# B&R Automation Studio project ProcessPointsTest
Automation Studio 4.11.6.26 SP; technology packages: mappMotion 5.23.1

## Configuration Config1

CPU PC_any, AutomationRuntime D4.92, Build 4.1.2, Safety 0.0, Vc V4.72.5

### Task classes (Cpu.sw)
```
Cyclic#1 (cycle 1600 us, tolerance 0 us):
  Program <- Program.prg
DataObjects: McAcpSys
NcDataObjects: McDriveLog
Binaries: arsvcreg, udbdef, McAcpDrv, arflatprv, arcoal, FWRules, TCData, McAcpSim, ashwd, ashwac, Points, User, Machine, sysconf, ShuttleCon, asfw, arconfig, ShuttleSim, iomap, Sectors, Role
Libraries: McBase, McAxis, McAcpTrak, MpBase, MpAxis, McAcpAx, standard, AsBrStr, runtime, asieccon, powerlnk, astime, fileio, sys_lib, asepl
```

### Hardware
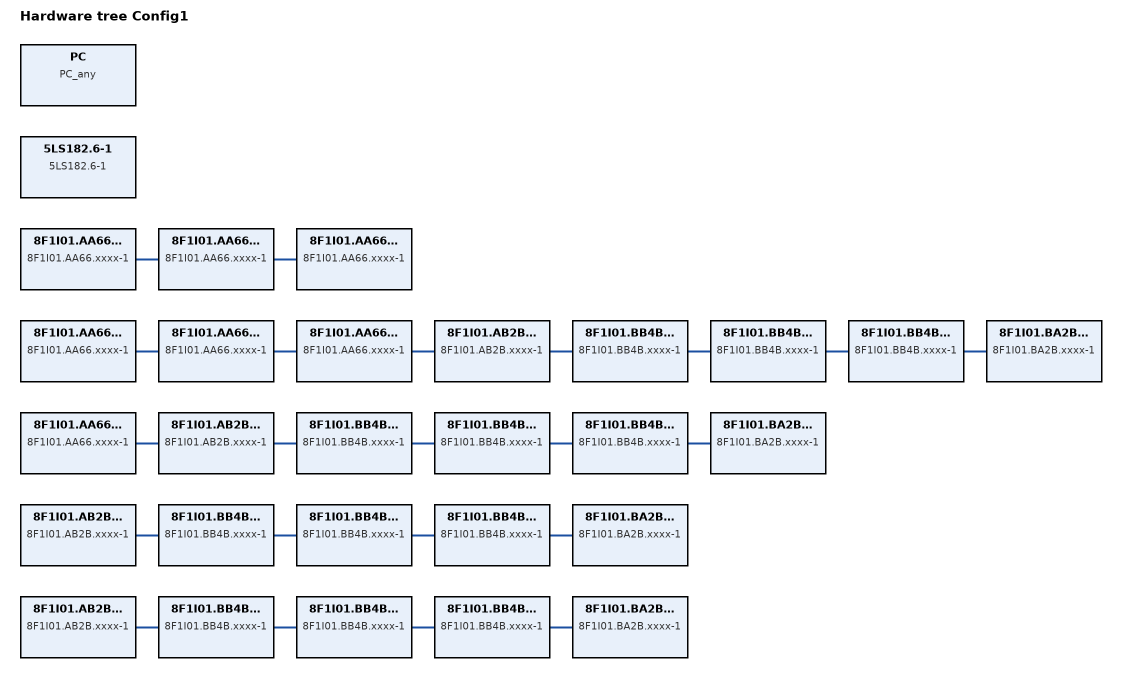
```
5LS182.6-1 : 5LS182.6-1 v1.3.1.0  [PLK2 -> 8F1I01.AA66.xxxx-1f.PLK3 [Cable Type=PowerlinkCable, Length=10, Version=1.0.0.3]; SL -> PC.SL1]
  Connector IF1:
    CycleTime = 800
  Supervision = off
8F1I01.AA66.xxxx-1 : 8F1I01.AA66.xxxx-1 v1.0.0.2  [PLK1 -> 8F1I01.BA2B.xxxx-1.PLK2 (NodeNumber=6) [Cable Type=PowerlinkCable, Length=10, Version=1.0.0.3]; PLK2 -> 8F1I01.AA66.xxxx-1a.PLK1 (NodeNumber=6) [Cable Type=PowerlinkCable, Length=10, Version=1.0.0.3]]
  DriveConfiguration:
    McTypeID = LLMConfig
  DriveConfiguration/Segment:
    Shape = STRAIGHT660
    SegmentReference = A06
    SegmentSectorDirection = Positive
    ElongationCompensation = UseAssemblySetting
    StopReaction = UseAssemblySetting
    SpeedFilter = UseAssemblySetting
    PositionControllerLagMonitor = UseAssemblySetting
8F1I01.AA66.xxxx-1a : 8F1I01.AA66.xxxx-1 v1.0.0.2  [PLK1 -> 8F1I01.AA66.xxxx-1.PLK2 (NodeNumber=7) [Cable Type=PowerlinkCable, Length=10, Version=1.0.0.3]; PLK2 -> 8F1I01.AA66.xxxx-1b.PLK1 (NodeNumber=7) [Cable Type=PowerlinkCable, Length=10, Version=1.0.0.3]]
  DriveConfiguration:
    McTypeID = LLMConfig
  DriveConfiguration/Segment:
    Shape = STRAIGHT660
    SegmentReference = A07
    SegmentSectorDirection = Positive
    ElongationCompensation = UseAssemblySetting
    StopReaction = UseAssemblySetting
    SpeedFilter = UseAssemblySetting
    PositionControllerLagMonitor = UseAssemblySetting
8F1I01.AA66.xxxx-1b : 8F1I01.AA66.xxxx-1 v1.0.0.2  [PLK1 -> 8F1I01.AA66.xxxx-1a.PLK2 (NodeNumber=8) [Cable Type=PowerlinkCable, Length=10, Version=1.0.0.3]]
  DriveConfiguration:
    McTypeID = LLMConfig
  DriveConfiguration/Segment:
    Shape = STRAIGHT660
    SegmentReference = A08
    SegmentSectorDirection = Positive
    ElongationCompensation = UseAssemblySetting
    StopReaction = UseAssemblySetting
    SpeedFilter = UseAssemblySetting
    PositionControllerLagMonitor = UseAssemblySetting
8F1I01.AA66.xxxx-1c : 8F1I01.AA66.xxxx-1 v1.0.0.2  [PLK1 -> 8F1I01.BA2B.xxxx-1a.PLK2 (NodeNumber=14) [Cable Type=PowerlinkCable, Length=10, Version=1.0.0.3]; PLK2 -> 8F1I01.AA66.xxxx-1d.PLK1 (NodeNumber=14) [Cable Type=PowerlinkCable, Length=10, Version=1.0.0.3]]
  DriveConfiguration:
    McTypeID = LLMConfig
  DriveConfiguration/Segment:
    Shape = STRAIGHT660
    SegmentReference = A14
    SegmentSectorDirection = Positive
    ElongationCompensation = UseAssemblySetting
    StopReaction = UseAssemblySetting
    SpeedFilter = UseAssemblySetting
    PositionControllerLagMonitor = UseAssemblySetting
8F1I01.AA66.xxxx-1d : 8F1I01.AA66.xxxx-1 v1.0.0.2  [PLK1 -> 8F1I01.AA66.xxxx-1c.PLK2 (NodeNumber=15) [Cable Type=PowerlinkCable, Length=10, Version=1.0.0.3]; PLK2 -> 8F1I01.AA66.xxxx-1e.PLK1 (NodeNumber=15) [Cable Type=PowerlinkCable, Length=10, Version=1.0.0.3]]
  DriveConfiguration:
    McTypeID = LLMConfig
  DriveConfiguration/Segment:
    Shape = STRAIGHT660
    SegmentReference = A15
    SegmentSectorDirection = Positive
    ElongationCompensation = UseAssemblySetting
    StopReaction = UseAssemblySetting
    SpeedFilter = UseAssemblySetting
    PositionControllerLagMonitor = UseAssemblySetting
8F1I01.AA66.xxxx-1e : 8F1I01.AA66.xxxx-1 v1.0.0.2  [PLK1 -> 8F1I01.AA66.xxxx-1d.PLK2 (NodeNumber=16) [Cable Type=PowerlinkCable, Length=10, Version=1.0.0.3]; PLK2 -> 8F1I01.AB2B.xxxx-1.PLK1 (NodeNumber=16) [Cable Type=PowerlinkCable, Length=10, Version=1.0.0.3]]
  DriveConfiguration:
    McTypeID = LLMConfig
  DriveConfiguration/Segment:
    Shape = STRAIGHT660
    SegmentReference = A16
    SegmentSectorDirection = Positive
    ElongationCompensation = UseAssemblySetting
    StopReaction = UseAssemblySetting
    SpeedFilter = UseAssemblySetting
    PositionControllerLagMonitor = UseAssemblySetting
8F1I01.AA66.xxxx-1f : 8F1I01.AA66.xxxx-1 v1.0.0.2  [PLK1 -> 8F1I01.BA2B.xxxx-1c.PLK2 (NodeNumber=17) [Cable Type=PowerlinkCable, Length=10, Version=1.0.0.3]; PLK2 -> 8F1I01.AB2B.xxxx-1b.PLK1 (NodeNumber=17) [Cable Type=PowerlinkCable, Length=10, Version=1.0.0.3]; PLK3 -> 5LS182.6-1.PLK2 (NodeNumber=17) [Cable Type=PowerlinkCable, Length=10, Version=1.0.0.3]]
  DriveConfiguration:
    McTypeID = LLMConfig
  DriveConfiguration/Segment:
    Shape = STRAIGHT660
    SegmentReference = B06
    SegmentSectorDirection = Positive
    ElongationCompensation = UseAssemblySetting
    StopReaction = UseAssemblySetting
    SpeedFilter = UseAssemblySetting
    PositionControllerLagMonitor = UseAssemblySetting
8F1I01.AB2B.xxxx-1 : 8F1I01.AB2B.xxxx-1 v1.0.0.2  [PLK1 -> 8F1I01.AA66.xxxx-1e.PLK2 (NodeNumber=1) [Cable Type=PowerlinkCable, Length=10, Version=1.0.0.3]; PLK2 -> 8F1I01.BB4B.xxxx-1.PLK1 (NodeNumber=1) [Cable Type=PowerlinkCable, Length=10, Version=1.0.0.3]; PLK3 -> 5LS182.6-1.IF1 (NodeNumber=1) [Cable Type=PowerlinkCable, Length=10, Version=1.0.0.3]]
  DriveConfiguration:
    McTypeID = LLMConfig
  DriveConfiguration/Segment:
    Shape = STRAIGHT105_TO_CIRCULAR
    SegmentReference = A01
    SegmentSectorDirection = Positive
    ElongationCompensation = UseAssemblySetting
    StopReaction = UseAssemblySetting
    SpeedFilter = UseAssemblySetting
    PositionControllerLagMonitor = UseAssemblySetting
8F1I01.AB2B.xxxx-1a : 8F1I01.AB2B.xxxx-1 v1.0.0.2  [PLK2 -> 8F1I01.BB4B.xxxx-1c.PLK1 (NodeNumber=9) [Cable Type=PowerlinkCable, Length=10, Version=1.0.0.3]]
  DriveConfiguration:
    McTypeID = LLMConfig
  DriveConfiguration/Segment:
    Shape = STRAIGHT105_TO_CIRCULAR
    SegmentReference = A09
    SegmentSectorDirection = Positive
    ElongationCompensation = UseAssemblySetting
    StopReaction = UseAssemblySetting
    SpeedFilter = UseAssemblySetting
    PositionControllerLagMonitor = UseAssemblySetting
8F1I01.AB2B.xxxx-1b : 8F1I01.AB2B.xxxx-1 v1.0.0.2  [PLK1 -> 8F1I01.AA66.xxxx-1f.PLK2 (NodeNumber=18) [Cable Type=PowerlinkCable, Length=10, Version=1.0.0.3]; PLK2 -> 8F1I01.BB4B.xxxx-1f.PLK1 (NodeNumber=18) [Cable Type=PowerlinkCable, Length=10, Version=1.0.0.3]]
  DriveConfiguration:
    McTypeID = LLMConfig
  DriveConfiguration/Segment:
    Shape = STRAIGHT105_TO_CIRCULAR
    SegmentReference = B07
    SegmentSectorDirection = Positive
    ElongationCompensation = UseAssemblySetting
    StopReaction = UseAssemblySetting
    SpeedFilter = UseAssemblySetting
    PositionControllerLagMonitor = UseAssemblySetting
8F1I01.AB2B.xxxx-1c : 8F1I01.AB2B.xxxx-1 v1.0.0.2  [PLK2 -> 8F1I01.BB4B.xxxx-1k.PLK1 (NodeNumber=27) [Cable Type=PowerlinkCable, Length=10, Version=1.0.0.3]]
  DriveConfiguration:
    McTypeID = LLMConfig
  DriveConfiguration/Segment:
    Shape = STRAIGHT105_TO_CIRCULAR
    SegmentReference = B01
    SegmentSectorDirection = Positive
    ElongationCompensation = UseAssemblySetting
    StopReaction = UseAssemblySetting
    SpeedFilter = UseAssemblySetting
    PositionControllerLagMonitor = UseAssemblySetting
8F1I01.BA2B.xxxx-1 : 8F1I01.BA2B.xxxx-1 v1.0.0.2  [PLK1 -> 8F1I01.BB4B.xxxx-1b.PLK2 (NodeNumber=5) [Cable Type=PowerlinkCable, Length=10, Version=1.0.0.3]; PLK2 -> 8F1I01.AA66.xxxx-1.PLK1 (NodeNumber=5) [Cable Type=PowerlinkCable, Length=10, Version=1.0.0.3]]
  DriveConfiguration:
    McTypeID = LLMConfig
  DriveConfiguration/Segment:
    Shape = CIRCULAR_TO_STRAIGHT105
    SegmentReference = A05
    SegmentSectorDirection = Positive
    ElongationCompensation = UseAssemblySetting
    StopReaction = UseAssemblySetting
    SpeedFilter = UseAssemblySetting
    PositionControllerLagMonitor = UseAssemblySetting
8F1I01.BA2B.xxxx-1a : 8F1I01.BA2B.xxxx-1 v1.0.0.2  [PLK1 -> 8F1I01.BB4B.xxxx-1e.PLK2 (NodeNumber=13) [Cable Type=PowerlinkCable, Length=10, Version=1.0.0.3]; PLK2 -> 8F1I01.AA66.xxxx-1c.PLK1 (NodeNumber=13) [Cable Type=PowerlinkCable, Length=10, Version=1.0.0.3]]
  DriveConfiguration:
    McTypeID = LLMConfig
  DriveConfiguration/Segment:
    Shape = CIRCULAR_TO_STRAIGHT105
    SegmentReference = A13
    SegmentSectorDirection = Positive
    ElongationCompensation = UseAssemblySetting
    StopReaction = UseAssemblySetting
    SpeedFilter = UseAssemblySetting
    PositionControllerLagMonitor = UseAssemblySetting
8F1I01.BA2B.xxxx-1b : 8F1I01.BA2B.xxxx-1 v1.0.0.2  [PLK1 -> 8F1I01.BB4B.xxxx-1h.PLK2 (NodeNumber=22) [Cable Type=PowerlinkCable, Length=10, Version=1.0.0.3]]
  DriveConfiguration:
    McTypeID = LLMConfig
  DriveConfiguration/Segment:
    Shape = CIRCULAR_TO_STRAIGHT105
    SegmentReference = B11
    SegmentSectorDirection = Positive
    ElongationCompensation = UseAssemblySetting
    StopReaction = UseAssemblySetting
    SpeedFilter = UseAssemblySetting
    PositionControllerLagMonitor = UseAssemblySetting
8F1I01.BA2B.xxxx-1c : 8F1I01.BA2B.xxxx-1 v1.0.0.2  [PLK1 -> 8F1I01.BB4B.xxxx-1i.PLK2 (NodeNumber=23) [Cable Type=PowerlinkCable, Length=10, Version=1.0.0.3]; PLK2 -> 8F1I01.AA66.xxxx-1f.PLK1 (NodeNumber=23) [Cable Type=PowerlinkCable, Length=10, Version=1.0.0.3]]
  DriveConfiguration:
    McTypeID = LLMConfig
  DriveConfiguration/Segment:
    Shape = CIRCULAR_TO_STRAIGHT105
    SegmentReference = B05
    SegmentSectorDirection = Positive
    ElongationCompensation = UseAssemblySetting
    StopReaction = UseAssemblySetting
    SpeedFilter = UseAssemblySetting
    PositionControllerLagMonitor = UseAssemblySetting
8F1I01.BB4B.xxxx-1 : 8F1I01.BB4B.xxxx-1 v1.0.0.2  [PLK1 -> 8F1I01.AB2B.xxxx-1.PLK2 (NodeNumber=2) [Cable Type=PowerlinkCable, Length=10, Version=1.0.0.3]; PLK2 -> 8F1I01.BB4B.xxxx-1a.PLK1 (NodeNumber=2) [Cable Type=PowerlinkCable, Length=10, Version=1.0.0.3]]
  DriveConfiguration:
    McTypeID = LLMConfig
  DriveConfiguration/Segment:
    Shape = CIRCULAR
    SegmentReference = A02
    SegmentSectorDirection = Positive
    ElongationCompensation = UseAssemblySetting
    StopReaction = UseAssemblySetting
    SpeedFilter = UseAssemblySetting
    PositionControllerLagMonitor = UseAssemblySetting
8F1I01.BB4B.xxxx-1a : 8F1I01.BB4B.xxxx-1 v1.0.0.2  [PLK1 -> 8F1I01.BB4B.xxxx-1.PLK2 (NodeNumber=3) [Cable Type=PowerlinkCable, Length=10, Version=1.0.0.3]; PLK2 -> 8F1I01.BB4B.xxxx-1b.PLK1 (NodeNumber=3) [Cable Type=PowerlinkCable, Length=10, Version=1.0.0.3]]
  DriveConfiguration:
    McTypeID = LLMConfig
  DriveConfiguration/Segment:
    Shape = CIRCULAR
    SegmentReference = A03
    SegmentSectorDirection = Positive
    ElongationCompensation = UseAssemblySetting
    StopReaction = UseAssemblySetting
    SpeedFilter = UseAssemblySetting
    PositionControllerLagMonitor = UseAssemblySetting
8F1I01.BB4B.xxxx-1b : 8F1I01.BB4B.xxxx-1 v1.0.0.2  [PLK1 -> 8F1I01.BB4B.xxxx-1a.PLK2 (NodeNumber=4) [Cable Type=PowerlinkCable, Length=10, Version=1.0.0.3]; PLK2 -> 8F1I01.BA2B.xxxx-1.PLK1 (NodeNumber=4) [Cable Type=PowerlinkCable, Length=10, Version=1.0.0.3]]
  DriveConfiguration:
    McTypeID = LLMConfig
  DriveConfiguration/Segment:
    Shape = CIRCULAR
    SegmentReference = A04
    SegmentSectorDirection = Positive
    ElongationCompensation = UseAssemblySetting
    StopReaction = UseAssemblySetting
    SpeedFilter = UseAssemblySetting
    PositionControllerLagMonitor = UseAssemblySetting
8F1I01.BB4B.xxxx-1c : 8F1I01.BB4B.xxxx-1 v1.0.0.2  [PLK1 -> 8F1I01.AB2B.xxxx-1a.PLK2 (NodeNumber=10) [Cable Type=PowerlinkCable, Length=10, Version=1.0.0.3]; PLK2 -> 8F1I01.BB4B.xxxx-1d.PLK1 (NodeNumber=10) [Cable Type=PowerlinkCable, Length=10, Version=1.0.0.3]]
  DriveConfiguration:
    McTypeID = LLMConfig
  DriveConfiguration/Segment:
    Shape = CIRCULAR
    SegmentReference = A10
    SegmentSectorDirection = Positive
    ElongationCompensation = UseAssemblySetting
    StopReaction = UseAssemblySetting
    SpeedFilter = UseAssemblySetting
    PositionControllerLagMonitor = UseAssemblySetting
8F1I01.BB4B.xxxx-1d : 8F1I01.BB4B.xxxx-1 v1.0.0.2  [PLK1 -> 8F1I01.BB4B.xxxx-1c.PLK2 (NodeNumber=11) [Cable Type=PowerlinkCable, Length=10, Version=1.0.0.3]; PLK2 -> 8F1I01.BB4B.xxxx-1e.PLK1 (NodeNumber=11) [Cable Type=PowerlinkCable, Length=10, Version=1.0.0.3]]
  DriveConfiguration:
    McTypeID = LLMConfig
  DriveConfiguration/Segment:
    Shape = CIRCULAR
    SegmentReference = A11
    SegmentSectorDirection = Positive
    ElongationCompensation = UseAssemblySetting
    StopReaction = UseAssemblySetting
    SpeedFilter = UseAssemblySetting
    PositionControllerLagMonitor = UseAssemblySetting
8F1I01.BB4B.xxxx-1e : 8F1I01.BB4B.xxxx-1 v1.0.0.2  [PLK1 -> 8F1I01.BB4B.xxxx-1d.PLK2 (NodeNumber=12) [Cable Type=PowerlinkCable, Length=10, Version=1.0.0.3]; PLK2 -> 8F1I01.BA2B.xxxx-1a.PLK1 (NodeNumber=12) [Cable Type=PowerlinkCable, Length=10, Version=1.0.0.3]]
  DriveConfiguration:
    McTypeID = LLMConfig
  DriveConfiguration/Segment:
    Shape = CIRCULAR
    SegmentReference = A12
    SegmentSectorDirection = Positive
    ElongationCompensation = UseAssemblySetting
    StopReaction = UseAssemblySetting
    SpeedFilter = UseAssemblySetting
    PositionControllerLagMonitor = UseAssemblySetting
8F1I01.BB4B.xxxx-1f : 8F1I01.BB4B.xxxx-1 v1.0.0.2  [PLK1 -> 8F1I01.AB2B.xxxx-1b.PLK2 (NodeNumber=19) [Cable Type=PowerlinkCable, Length=10, Version=1.0.0.3]; PLK2 -> 8F1I01.BB4B.xxxx-1g.PLK1 (NodeNumber=19) [Cable Type=PowerlinkCable, Length=10, Version=1.0.0.3]]
  DriveConfiguration:
    McTypeID = LLMConfig
  DriveConfiguration/Segment:
    Shape = CIRCULAR
    SegmentReference = B08
    SegmentSectorDirection = Positive
    ElongationCompensation = UseAssemblySetting
    StopReaction = UseAssemblySetting
    SpeedFilter = UseAssemblySetting
    PositionControllerLagMonitor = UseAssemblySetting
8F1I01.BB4B.xxxx-1g : 8F1I01.BB4B.xxxx-1 v1.0.0.2  [PLK1 -> 8F1I01.BB4B.xxxx-1f.PLK2 (NodeNumber=20) [Cable Type=PowerlinkCable, Length=10, Version=1.0.0.3]; PLK2 -> 8F1I01.BB4B.xxxx-1h.PLK1 (NodeNumber=20) [Cable Type=PowerlinkCable, Length=10, Version=1.0.0.3]]
  DriveConfiguration:
    McTypeID = LLMConfig
  DriveConfiguration/Segment:
    Shape = CIRCULAR
    SegmentReference = B09
    SegmentSectorDirection = Positive
    ElongationCompensation = UseAssemblySetting
    StopReaction = UseAssemblySetting
    SpeedFilter = UseAssemblySetting
    PositionControllerLagMonitor = UseAssemblySetting
8F1I01.BB4B.xxxx-1h : 8F1I01.BB4B.xxxx-1 v1.0.0.2  [PLK1 -> 8F1I01.BB4B.xxxx-1g.PLK2 (NodeNumber=21) [Cable Type=PowerlinkCable, Length=10, Version=1.0.0.3]; PLK2 -> 8F1I01.BA2B.xxxx-1b.PLK1 (NodeNumber=21) [Cable Type=PowerlinkCable, Length=10, Version=1.0.0.3]]
  DriveConfiguration:
    McTypeID = LLMConfig
  DriveConfiguration/Segment:
    Shape = CIRCULAR
    SegmentReference = B10
    SegmentSectorDirection = Positive
    ElongationCompensation = UseAssemblySetting
    StopReaction = UseAssemblySetting
    SpeedFilter = UseAssemblySetting
    PositionControllerLagMonitor = UseAssemblySetting
8F1I01.BB4B.xxxx-1i : 8F1I01.BB4B.xxxx-1 v1.0.0.2  [PLK1 -> 8F1I01.BB4B.xxxx-1j.PLK2 (NodeNumber=24) [Cable Type=PowerlinkCable, Length=10, Version=1.0.0.3]; PLK2 -> 8F1I01.BA2B.xxxx-1c.PLK1 (NodeNumber=24) [Cable Type=PowerlinkCable, Length=10, Version=1.0.0.3]]
  DriveConfiguration:
    McTypeID = LLMConfig
  DriveConfiguration/Segment:
    Shape = CIRCULAR
    SegmentReference = B04
    SegmentSectorDirection = Positive
    ElongationCompensation = UseAssemblySetting
    StopReaction = UseAssemblySetting
    SpeedFilter = UseAssemblySetting
    PositionControllerLagMonitor = UseAssemblySetting
8F1I01.BB4B.xxxx-1j : 8F1I01.BB4B.xxxx-1 v1.0.0.2  [PLK1 -> 8F1I01.BB4B.xxxx-1k.PLK2 (NodeNumber=25) [Cable Type=PowerlinkCable, Length=10, Version=1.0.0.3]; PLK2 -> 8F1I01.BB4B.xxxx-1i.PLK1 (NodeNumber=25) [Cable Type=PowerlinkCable, Length=10, Version=1.0.0.3]]
  DriveConfiguration:
    McTypeID = LLMConfig
  DriveConfiguration/Segment:
    Shape = CIRCULAR
    SegmentReference = B03
    SegmentSectorDirection = Positive
    ElongationCompensation = UseAssemblySetting
    StopReaction = UseAssemblySetting
    SpeedFilter = UseAssemblySetting
    PositionControllerLagMonitor = UseAssemblySetting
8F1I01.BB4B.xxxx-1k : 8F1I01.BB4B.xxxx-1 v1.0.0.2  [PLK1 -> 8F1I01.AB2B.xxxx-1c.PLK2 (NodeNumber=26) [Cable Type=PowerlinkCable, Length=10, Version=1.0.0.3]; PLK2 -> 8F1I01.BB4B.xxxx-1j.PLK1 (NodeNumber=26) [Cable Type=PowerlinkCable, Length=10, Version=1.0.0.3]]
  DriveConfiguration:
    McTypeID = LLMConfig
  DriveConfiguration/Segment:
    Shape = CIRCULAR
    SegmentReference = B02
    SegmentSectorDirection = Positive
    ElongationCompensation = UseAssemblySetting
    StopReaction = UseAssemblySetting
    SpeedFilter = UseAssemblySetting
    PositionControllerLagMonitor = UseAssemblySetting
PC : PC_any v1.1.1.0 (OrderNumber=PC)
  ConfigurationID = ProcessPointsTest_Config1
  SystemTick = 800
  Cyclic1Duration = 1600
  Cyclic1Tolerance = 0
  FileDevice1
  FileDeviceName1 = USER
  FileDevicePath1 = USER_PATH
  FileDevice2
  FileDeviceName2 = SvgData
  FileDevicePath2 = C:\SceneViewerFiles\ProcessPointsTest
  ActivateOpcUa = 1
  OpcUaInformationModels_PV_Version = 1
```

### Machine.assembly - PC/mappMotion/Machine.assembly
```
Element gAssembly_1 (Type=assembly)
  Tracks:
    TrackSeparation = 0.030
    Track[1]:
      Segments:
        SegmentRef[1] = ::A01
        SegmentRef[2] = ::A02
        SegmentRef[3] = ::A03
        SegmentRef[4] = ::A04
        SegmentRef[5] = ::A05
        SegmentRef[6] = ::A06
        SegmentRef[7] = ::A07
        SegmentRef[8] = ::A08
        SegmentRef[9] = ::A09
        SegmentRef[10] = ::A10
        SegmentRef[11] = ::A11
        SegmentRef[12] = ::A12
        SegmentRef[13] = ::A13
        SegmentRef[14] = ::A14
        SegmentRef[15] = ::A15
        SegmentRef[16] = ::A16
      Position = Absolute
        SegmentCountDirection = RightToLeft
        Translation:
          X = 0.0
          Y = 0.0
          Z = 0.0
        Orientation:
          Angle1 = 0.0
          Angle2 = 0.0
          Angle3 = 0.0
    Track[2]:
      Segments:
        SegmentRef[1] = ::B01
        SegmentRef[2] = ::B02
        SegmentRef[3] = ::B03
        SegmentRef[4] = ::B04
        SegmentRef[5] = ::B05
        SegmentRef[6] = ::B06
        SegmentRef[7] = ::B07
        SegmentRef[8] = ::B08
        SegmentRef[9] = ::B09
        SegmentRef[10] = ::B10
        SegmentRef[11] = ::B11
      Position = RelativeToOne
        TrackSegmentPosition:
          SegmentRef = ::B01
        Base:
          SegmentRef = ::A05
          PositionRelativeTo = FromEnd
  CommonSegmentSettings:
    SegmentSimulationOnPLC = Off
    CoggingCompensation = Active
      UpperVelLimit = 0.5
    ElongationCompensation = Inactive
    StopReaction = InductionHalt
    SpeedFilter = NotUsed
    ControllerParameters:
      DefaultParameter:
        Controller:
          Position:
            ProportionalGain = 0.0
          Speed:
            ProportionalGain = 0.0
            IntegrationTime = 0.0
          FeedForward:
            TotalMass = 0.0
            ForcePositive = 0.0
            ForceNegative = 0.0
            SpeedForceFactor = 0.0
            ForceLoad = 0.0
        MovementErrorLimits:
          PositionError = 0.004
          VelocityError = 1.2
        Diverter:
          ForceOverride = 1.0
      AdditionalParameterSets = NotUsed
    ScopeOfErrorReaction = Assembly
    ShuttleIdentificationTime = 0
    PositionControllerLagMonitor = Inactive
    Diverter:
      DiverterWeakEndOverrideFactor = 1.0
      DiverterStrenEndOverrideFactor = 1.0
  Shuttles:
    MaxShuttleCount = 50
    MaxShuttleCommandCount = 0
    Deceleration = 0.0
    UseConvoys = Inactive
    DistanceReserve:
      Collision = 0.002
      ErrorStop = 0.006
    ShuttleStereotypes:
      ShuttleStRef[1] = ShuttleStereotype_1
    MagnetPlateConfigurations:
      ShuttleType[1] = 8F1SA.100.xxxxxx-x
    CollisionAvoidance:
      Strategy = Constant
      Exclusion = NotUsed
      MaximumModelDimensions:
        Length:
          ExtentToFront = 0.025
          ExtentToBack = 0.025
        Width:
          Width = 0.046
    Coupling:
      CouplingFeature:
        EliminateShuttleToShuttleDelay = FALSE
  Visualization:
    MonitoringPv
    ProcessingTaskClass = 4
  Alarms = None
```

### Points.processpointlist - PC/mappMotion/Points.processpointlist
```
Element ProcessPointList_1 (Type=processpointlist)
  ProcessPoint[0]:
    Name = PPThroughput
    SectorRef = SectorMainLoop
    Position = 0.81
    TriggerEventBufferSize = 10
    BarrierFunctionality = Off
  ProcessPoint[1]:
    Name = PPBuffer
    SectorRef = SectorBuffer
    Position = 0.2
    TriggerEventBufferSize = 10
    BarrierFunctionality = Off
  ProcessPoint[2]:
    Name = PPStation0
    SectorRef = SectorWorkZone
    TriggerEventBufferSize = 10
    BarrierFunctionality = On
  ProcessPoint[3]:
    Name = PPStation1
    SectorRef = SectorWorkZone
    Position = 0.495
    TriggerEventBufferSize = 10
    BarrierFunctionality = Off
  ProcessPoint[4]:
    Name = PPStation2
    SectorRef = SectorWorkZone
    Position = 0.99
    TriggerEventBufferSize = 10
    BarrierFunctionality = Off
  ProcessPoint[5]:
    Name = PPStation3
    SectorRef = SectorWorkZone
    Position = 1.485
    TriggerEventBufferSize = 10
    BarrierFunctionality = Off
  ProcessPoint[6]:
    Name = PPStation4
    SectorRef = SectorWorkZone
    Position = 1.98
    TriggerEventBufferSize = 10
    BarrierFunctionality = Off
  ProcessPoint[7]:
    Name = PPMaintenancePoint
    SectorRef = SectorMaintenancePoint
    Position = 0.33
    TriggerEventBufferSize = 10
    BarrierFunctionality = Off
  ProcessPoint[8]:
    Name = PPStation0TrgPoint
    SectorRef = BarrierTrgPoint
    Position = 0.026
    PositionRelativeTo = FromEnd
    TriggerEventBufferSize = 10
    BarrierFunctionality = Off
```

### Sectors.sector - PC/mappMotion/Sectors.sector
```
Element MainLoop (Type=sector)
  Type = Composed
    StartSegment:
      SegmentRef = ::A01
    IntermediateSegments:
      SegmentRef[1] = ::A02
      SegmentRef[2] = ::A03
      SegmentRef[3] = ::A04
      SegmentRef[4] = ::A05
      SegmentRef[5] = ::A06
      SegmentRef[6] = ::A07
      SegmentRef[7] = ::A08
      SegmentRef[8] = ::A09
      SegmentRef[9] = ::A10
      SegmentRef[10] = ::A11
      SegmentRef[11] = ::A12
      SegmentRef[12] = ::A13
      SegmentRef[13] = ::A14
      SegmentRef[14] = ::A15
    EndSegment:
      SegmentRef = ::A16
      PositionRelativeTo = FromEnd
  Alarms = None
Element MaintLoop (Type=sector)
  Type = Composed
    StartSegment:
      SegmentRef = ::B11
    IntermediateSegments:
      SegmentRef[1] = ::B10
      SegmentRef[2] = ::B09
      SegmentRef[3] = ::B08
      SegmentRef[4] = ::B07
      SegmentRef[5] = ::B06
      SegmentRef[6] = ::B05
      SegmentRef[7] = ::B04
      SegmentRef[8] = ::B03
      SegmentRef[9] = ::B02
    EndSegment:
      SegmentRef = ::B01
      PositionRelativeTo = FromEnd
  Alarms = None
Element Barrier (Type=sector)
  Type = Composed
    StartSegment:
      SegmentRef = ::A08
    EndSegment:
      SegmentRef = ::A08
      PositionRelativeTo = FromEnd
  Alarms = None
Element ProcessPoints (Type=sector)
  Type = Composed
    StartSegment:
      SegmentRef = ::A14
    IntermediateSegments:
      SegmentRef[1] = ::A15
    EndSegment:
      SegmentRef = ::A16
      PositionRelativeTo = FromEnd
  Alarms = None
Element MaintPoint (Type=sector)
  Type = Composed
    StartSegment:
      SegmentRef = ::B06
    EndSegment:
      SegmentRef = ::B06
      PositionRelativeTo = FromEnd
  Alarms = None
```

### ShuttleCon.shuttlestereotype - PC/mappMotion/ShuttleCon.shuttlestereotype
```
Element ShuttleStereotype_1 (Type=shuttlestereotype)
  MeasurementUnit = 5067858
  MeasurementResolution = 0.00001
  MovementLimits = Internal
    VelocityIsReadOnly = 0
    Velocity:
      Velocity = 5.5
    AccelerationIsReadOnly = 0
    Acceleration:
      Acceleration = 100.0
    DecelerationIsReadOnly = 0
    Deceleration:
      Deceleration = 100.0
    UpdateMode = Immediately
  JerkFilter = Used
    JerkTime = 0.02
  UserData:
    Size = 0
  StateTransitions:
    AutomaticRecontrol = Active
```

### ShuttleSim.assemblyfeature - PC/mappMotion/ShuttleSim.assemblyfeature
```
Element ShuttleSim (Type=assemblyfeature)
  Type = InitShuttleSim
    InitShuttleSim[1]:
      SectorRef = MainLoop
      Orientation = Positive
      ShuttleDefinition = ShuttleSetDefinition
        StartPosition = 0.1
        NumberOfShuttles = 15
        DistnaceBetweenShuttles = 0.15
```

## Logical view

Binary libraries used (declarations not repeated): operator, runtime, astime, AsIecCon, McBase 5.23.1, McAxis 5.23.1, McAcpTrak 5.23.1, MpBase, MpAxis 5.23.1, McAcpAx 5.23.1, standard, AsBrStr

### Global.typ - Global data types
```iecst
(*Structures*)

TYPE
	TrakAssemblyControlType : 	STRUCT
		Command : TrakAssemblyCommandType;
		Parameter : TrakAssemblyParameterType;
		Status : TrakAssemblyStatusType;
		ShuttleCnt : UINT;
	END_STRUCT;
	TrakAssemblyCommandType : 	STRUCT
		Power : BOOL;
		StartMovement : BOOL;
		StopMovement : BOOL;
		Reset : BOOL;
	END_STRUCT;
	TrakAssemblyParameterType : 	STRUCT
		Velocity : REAL := 2.0;
		Acceleration : REAL := 20.0;
		Deceleration : REAL := 20.0;
	END_STRUCT;
	TrakAssemblyStatusType : 	STRUCT
		Disabled : BOOL;
		Ready : BOOL;
		Homing : BOOL;
		Stopping : BOOL;
		ErrorStop : BOOL;
	END_STRUCT;
	ShuttleControlType : 	STRUCT
		Axis : McAxisType;
		RoutedMoveAbs : MC_BR_RoutedMoveAbs_AcpTrak;
		State : ShuttleStateEnum := RTE_TO_BUFFER;
	END_STRUCT;
	ProcessPointLocations : 	STRUCT
		THROUGHPUT : REAL;
		BUFFER : REAL;
		WORK_ZONE : REAL;
		WORK_ZONE_TRG_POINT : REAL;
		WORK_STATION1 : REAL;
		WORK_STATION2 : REAL;
		WORK_STATION3 : REAL;
		WORK_STATION4 : REAL;
		MAINTENANCE_POINT : REAL;
	END_STRUCT;
END_TYPE

(*Enumerations*)

TYPE
	ShuttleStateEnum :
		(
		RTE_TO_BUFFER := 10,
		AT_BUFFER := 15,
		RTE_TO_STATION_1 := 20,
		AT_STATION_1 := 25,
		RTE_TO_STATION_2 := 30,
		AT_STATION_2 := 35,
		RTE_TO_STATION_3 := 40,
		AT_STATION_3 := 45,
		RTE_TO_STATION_4 := 50,
		AT_STATION_4 := 55,
		RTE_TO_MAINT := 60,
		AT_MAINT := 65
		);
	ProcessPointStateEnum :
		(
		WAIT,
		DO_NOTHING,
		DIRECTION_CHECK,
		PROCESS,
		SEND_SHUTTLE
		);
END_TYPE
```

### Global.var - Global variables
```iecst
(*Function blocks*)
VAR
	gTrakAsm : TrakAssemblyControlType;
	gRoutedMoveVel : MC_BR_RoutedMoveVel_AcpTrak;
	gThroughputTimer : TON;
END_VAR
(*Structures*)
VAR
	gShuttleList : ARRAY[1..gMAX_SHUTTLE_CNT] OF ShuttleControlType;
END_VAR
(*Variables*)
VAR
	gStation1EventCount : UINT;
	gStation1ReadyForShuttle : BOOL := TRUE;
	gStation2ReadyForShuttle : BOOL := TRUE;
	gStation3ReadyForShuttle : BOOL := TRUE;
	gStation4ReadyForShuttle : BOOL := TRUE;
	gCurrentThroughput : INT := 0;
END_VAR
(*Constants*)
VAR CONSTANT
	gMAX_SHUTTLE_CNT : USINT := 50;
	gMAX_SHUTTLES_TO_STATION_1 : UINT := 3;
	gTHROUGHPUT_TIMER_LENGTH : TIME := T#60s;
END_VAR
VAR
	gMAINTENCANCE_TIMER_LENGTH : TIME := T#5s;
	gPROCESS_TIMER_LENGTH : TIME := T#2s;
	gPROCESS_POINT_LOCATIONS : ProcessPointLocations := (THROUGHPUT:=0.81,BUFFER:=0.2,WORK_ZONE:=0.0,WORK_ZONE_TRG_POINT:=0.026,WORK_STATION1:=0.495,WORK_STATION2:=0.99,WORK_STATION3:=1.485,WORK_STATION4:=1.98,MAINTENANCE_POINT:=0.33);
END_VAR
```


### Program Logical/Program (IEC)

#### Main.st - Init, cyclic, exit code
```iecst
PROGRAM _INIT
	(* Initializing function blocks and their inputs *)
	AsmPowerOn.Assembly := ADR(gAssembly_1);
	AsmPowerOff.Assembly := ADR(gAssembly_1);
	AsmGetShuttle.Assembly := ADR(gAssembly_1);
	AsmStop.Assembly := ADR(gAssembly_1);
	AsmStop.StopMode := mcSTOPMODE_JERK_LIMIT;
	AsmReadStatus.Assembly := ADR(gAssembly_1);
	AsmReadStatus.Enable := TRUE;

	(* Initializing parameters for shuttle movements *)
	gTrakAsm.Parameter := SHUTTLE_PARAMETERS;
END_PROGRAM

PROGRAM _CYCLIC
	IF gTrakAsm.Status.ErrorStop THEN
		Step := ERROR;
	END_IF

	CASE Step OF

		POWER_OFF:
			IF gTrakAsm.Status.Disabled THEN
				AsmPowerOff.Execute := FALSE;
				Step := POWERED_OFF;
			END_IF

		WAIT_POWER_OFF:

		POWERED_OFF:
			IF gTrakAsm.Command.Power AND gTrakAsm.Status.Disabled THEN
				AsmPowerOn.Execute := TRUE;
				Step := POWER_ON;
			END_IF

		POWER_ON:
			IF AsmPowerOn.Done AND gTrakAsm.Status.Ready THEN
				AsmPowerOn.Execute := FALSE;
				FOR i := 1 TO gMAX_SHUTTLE_CNT DO
					brsmemset(ADR(gShuttleList[i].Axis), 0, SIZEOF(gShuttleList[i].Axis));
				END_FOR
				CurrentShuttleNumber := 1;
				Step := GET_SHUTTLE;
			END_IF

		WAIT_POWER_ON:

		GET_SHUTTLE:
			AsmGetShuttle.Enable := TRUE;

			IF AsmGetShuttle.Valid THEN
				(* There are no shuttles on the assembly. *)
				IF AsmGetShuttle.TotalCount = 0 THEN
					gTrakAsm.ShuttleCnt := 0;
					AsmGetShuttle.Enable := FALSE;
					AsmGetShuttle.Next := FALSE;

					Step := READY;
                (* As soon as the next shuttle has been output by the function block, RemainingCount
                   is reduced and this condition becomes true. *)
				ELSIF (AsmGetShuttle.RemainingCount <> (AsmGetShuttle.TotalCount - CurrentShuttleNumber)) THEN
					CurrentShuttleNumber := CurrentShuttleNumber + 1;
					AsmGetShuttle.Next := FALSE;
				ELSE
					(* Store all axis references in an array for global movement commands. *)
					gShuttleList[CurrentShuttleNumber].Axis := AsmGetShuttle.Axis;
					(* Get next shuttle reference with positive edge on .Next. *)
					AsmGetShuttle.Next := TRUE;

					(* All shuttles have been stored. *)
					IF (AsmGetShuttle.RemainingCount = 0) THEN
						gTrakAsm.ShuttleCnt := AsmGetShuttle.TotalCount;
						AsmGetShuttle.Enable := FALSE;
						AsmGetShuttle.Next := FALSE;

						Step := READY;
					END_IF
				END_IF
			END_IF

		READY:
			IF NOT gTrakAsm.Command.Power THEN
				AsmPowerOff.Execute := TRUE;
				Step := POWER_OFF;
			ELSIF gTrakAsm.Command.StartMovement AND gTrakAsm.ShuttleCnt > 0 THEN
				gTrakAsm.Command.StartMovement := FALSE;
				Step := START_MOVEMENT;
			END_IF

		START_MOVEMENT:
			FOR CurrentShuttleNumber := 1 TO gTrakAsm.ShuttleCnt DO
				gShuttleList[CurrentShuttleNumber].RoutedMoveAbs.Axis := ADR(gShuttleList[CurrentShuttleNumber].Axis);
				gShuttleList[CurrentShuttleNumber].RoutedMoveAbs.Sector := ADR(SectorBuffer);
				gShuttleList[CurrentShuttleNumber].RoutedMoveAbs.Position := gPROCESS_POINT_LOCATIONS.BUFFER;
				gShuttleList[CurrentShuttleNumber].RoutedMoveAbs.Velocity := gTrakAsm.Parameter.Velocity;
				gShuttleList[CurrentShuttleNumber].RoutedMoveAbs.Acceleration := gTrakAsm.Parameter.Acceleration;
				gShuttleList[CurrentShuttleNumber].RoutedMoveAbs.Deceleration := gTrakAsm.Parameter.Deceleration;
				gShuttleList[CurrentShuttleNumber].RoutedMoveAbs.Jerk := 0.0;
				gShuttleList[CurrentShuttleNumber].RoutedMoveAbs.BufferMode := mcABORTING;
				gShuttleList[CurrentShuttleNumber].RoutedMoveAbs.Execute := TRUE;
			END_FOR

			Step := WAIT_START_MOVEMENT;

		WAIT_START_MOVEMENT:
			FOR CurrentShuttleNumber := 1 TO gTrakAsm.ShuttleCnt DO
				gShuttleList[CurrentShuttleNumber].RoutedMoveAbs.Execute := FALSE;
			END_FOR

			gThroughputTimer.IN := TRUE;
			gThroughputTimer.PT := gTHROUGHPUT_TIMER_LENGTH;

			Step := MOVING;

		MOVING:
			IF gTrakAsm.Command.StopMovement THEN
				gTrakAsm.Command.StopMovement := FALSE;
				Step := STOPPING;
			END_IF

		STOPPING:
			FOR CurrentShuttleNumber := 1 TO gMAX_SHUTTLE_CNT DO
				gShuttleList[CurrentShuttleNumber].RoutedMoveAbs.Execute := FALSE;
			END_FOR
			AsmStop.Execute := TRUE;

			IF AsmStop.Done THEN
				AsmStop.Execute := FALSE;
				Step := READY;
			END_IF

		WAIT_STOPPING:

		ERROR:

		RESET:

	END_CASE

	(* Read assembly status cyclically to assembly interface. *)
	gTrakAsm.Status.Disabled := AsmReadStatus.AssemblyDisabled;
	gTrakAsm.Status.Ready := AsmReadStatus.AssemblyReady;
	gTrakAsm.Status.Homing := AsmReadStatus.AssemblyHoming;
	gTrakAsm.Status.Stopping := AsmReadStatus.AssemblyStopping;
	gTrakAsm.Status.ErrorStop := AsmReadStatus.AssemblyErrorStop;

	(* Calling function blocks *)
	AsmPowerOn();
	AsmPowerOff();
	AsmGetShuttle();
	AsmStop();
	AsmReadStatus();
	FOR i := 1 TO gMAX_SHUTTLE_CNT DO
		IF gShuttleList[i].Axis.controlif <> 0 THEN
			gShuttleList[i].RoutedMoveAbs();
		END_IF
	END_FOR
	gThroughputTimer();

	gCurrentThroughput;
END_PROGRAM

PROGRAM _EXIT
	(* Insert code here *)

END_PROGRAM
```

#### Types.typ - Local data types
```iecst
TYPE
	ProcessPointsFubsType : 	STRUCT
		Command : MC_BR_BarrierCommand_AcpTrak;
		BarrierReadInfo : MC_BR_BarrierReadInfo_AcpTrak;
		GetShuttle : MC_BR_BarrierGetShuttle_AcpTrak;
		ElasticMoveAbs : MC_BR_ElasticMoveAbs_AcpTrak;
		RoutedMoveVel : MC_BR_RoutedMoveVel_AcpTrak;
		RoutedMoveAbs : MC_BR_RoutedMoveAbs_AcpTrak;
		TrgEnable : MC_BR_TrgPointEnable_AcpTrak;
		TrgGetInfo : MC_BR_TrgPointGetInfo_AcpTrak;
		Timer : TON := (PT:=T#2s);
		Step : ProcessPointStateEnum;
		Shuttle : McAxisType;
		ReadyForShuttle : BOOL := TRUE;
	END_STRUCT;
	StateMachineEnum :
		(
		POWER_OFF := 10,
		WAIT_POWER_OFF := 20,
		POWERED_OFF := 30,
		POWER_ON := 40,
		WAIT_POWER_ON := 50,
		GET_SHUTTLE := 60,
		READY := 70,
		START_MOVEMENT := 80,
		WAIT_START_MOVEMENT := 90,
		MOVING := 100,
		STOPPING := 110,
		WAIT_STOPPING := 120,
		ERROR := 500,
		RESET := 510
		);
END_TYPE
```

#### Variables.var - Local variables
```iecst
(*Function Blocks*)
VAR
	AsmPowerOn : MC_BR_AsmPowerOn_AcpTrak;
	AsmPowerOff : MC_BR_AsmPowerOff_AcpTrak;
	AsmGetShuttle : MC_BR_AsmGetShuttle_AcpTrak;
	AsmStop : MC_BR_AsmStop_AcpTrak;
	AsmReadStatus : MC_BR_AsmReadStatus_AcpTrak;
END_VAR
(*Structures*)
(*Constants*)
VAR CONSTANT
	SHUTTLE_PARAMETERS : TrakAssemblyParameterType := (Velocity:=2.0,Acceleration:=20.0,Deceleration:=20.0);
END_VAR
(*Variables*)
VAR
	Step : StateMachineEnum := POWERED_OFF;
	i : UINT;
	CurrentShuttleNumber : UINT;
	ShuttlesToStation1 : UINT;
END_VAR
```

#### ActBufferBarrier.st
```iecst
ACTION ActBufferBarrier:

	CASE BufferBarrier.Step OF
		WAIT:
			BufferBarrier.RoutedMoveAbs.Execute := FALSE;

			ShuttlesToStation1 := 0;
			FOR i := 1 TO gMAX_SHUTTLE_CNT DO
				IF gShuttleList[i].State = RTE_TO_STATION_1 THEN
					ShuttlesToStation1 := ShuttlesToStation1 + 1;
				END_IF
			END_FOR

			IF BufferBarrier.TrgEnable.EventCount > 0 AND ShuttlesToStation1 < MAX_SHUTTLES_TO_STATION_1 THEN
				BufferBarrier.TrgGetInfo.Execute := TRUE;
				BufferBarrier.Step := DIRECTION_CHECK;
			END_IF

		DIRECTION_CHECK:
			IF BufferBarrier.TrgGetInfo.TrgPointInfo.Event = mcACPTRAK_TP_PASSED_POSITIVE THEN
				BufferBarrier.Shuttle := BufferBarrier.TrgGetInfo.TrgPointInfo.Axis;

				FOR i := 1 TO gMAX_SHUTTLE_CNT DO
					IF BufferBarrier.Shuttle.controlif = gShuttleList[i].Axis.controlif THEN
						gShuttleList[i].State := AT_BUFFER;
					END_IF
				END_FOR

				BufferBarrier.TrgGetInfo.Execute := FALSE;
				BufferBarrier.Step := SEND_SHUTTLE;
			ELSE
				BufferBarrier.TrgGetInfo.Execute := FALSE;
				BufferBarrier.Step := WAIT;
			END_IF

		SEND_SHUTTLE:
			BufferBarrier.RoutedMoveAbs.Axis := ADR(BufferBarrier.Shuttle);
			BufferBarrier.RoutedMoveAbs.Sector := ADR(SectorWorkZone);
			BufferBarrier.RoutedMoveAbs.Position := 0.0;
			BufferBarrier.RoutedMoveAbs.Velocity := gTrakAsm.Parameter.Velocity;
			BufferBarrier.RoutedMoveAbs.Acceleration := gTrakAsm.Parameter.Acceleration;
			BufferBarrier.RoutedMoveAbs.Deceleration := gTrakAsm.Parameter.Deceleration;
			BufferBarrier.RoutedMoveAbs.Jerk := 0.0;
			BufferBarrier.RoutedMoveAbs.BufferMode := mcABORTING;
			BufferBarrier.RoutedMoveAbs.Execute := TRUE;

			FOR i := 1 TO gMAX_SHUTTLE_CNT DO
				IF BufferBarrier.Shuttle.controlif = gShuttleList[i].Axis.controlif THEN
					gShuttleList[i].State := RTE_TO_STATION_1;
				END_IF
			END_FOR

			BufferBarrier.Step := WAIT;

	END_CASE

	BufferBarrier.Command();
	BufferBarrier.RoutedMoveAbs();
	BufferBarrier.TrgEnable();
	BufferBarrier.TrgGetInfo();
END_ACTION
```

#### ActWorkZone.st
```iecst
ACTION ActWorkZone:

	CASE WorkZone.Step OF
		WAIT:
			WorkZone.Command.Command := mcACPTRAK_BARRIER_CLOSE;
			WorkZone.Command.Execute := TRUE;

			IF WorkZone.TrgEnable.EventCount > 0 AND WorkStation1.ReadyForShuttle THEN
				WorkZone.Command.Execute := FALSE;
				WorkZone.TrgGetInfo.Execute := TRUE;
				WorkZone.Step := DIRECTION_CHECK;
			END_IF

		DIRECTION_CHECK:
			IF WorkZone.TrgGetInfo.TrgPointInfo.Event = mcACPTRAK_TP_PASSED_POSITIVE THEN
				WorkZone.Shuttle := WorkZone.TrgGetInfo.TrgPointInfo.Axis;
				WorkZone.TrgGetInfo.Execute := FALSE;
				WorkZone.Step := PROCESS;
			ELSE
				WorkZone.TrgGetInfo.Execute := FALSE;
				WorkZone.Step := WAIT;
			END_IF

		PROCESS:
			IF WorkStation1.TrgEnable.EventCount = 0 THEN
				WorkZone.Step := SEND_SHUTTLE;
			END_IF

		SEND_SHUTTLE:
			WorkZone.RoutedMoveAbs.Axis := ADR(WorkZone.Shuttle);
			WorkZone.RoutedMoveAbs.Sector := ADR(SectorWorkZone);
			WorkZone.RoutedMoveAbs.Position := 0.495;
			WorkZone.RoutedMoveAbs.Velocity := gTrakAsm.Parameter.Velocity;
			WorkZone.RoutedMoveAbs.Acceleration := gTrakAsm.Parameter.Acceleration;
			WorkZone.RoutedMoveAbs.Deceleration := gTrakAsm.Parameter.Deceleration;
			WorkZone.RoutedMoveAbs.Jerk := 0.0;
			WorkZone.RoutedMoveAbs.BufferMode := mcABORTING;
			WorkZone.RoutedMoveAbs.Execute := TRUE;

			WorkZone.Command.Command := mcACPTRAK_BARRIER_ADD_TICKETS;
			WorkZone.Command.AdvancedParameters.TicketCount := 1;
			WorkZone.Command.Execute := TRUE;

			IF WorkZone.Command.Done THEN
				WorkStation1.ReadyForShuttle := FALSE;
				WorkZone.Command.Execute := FALSE;
				WorkZone.RoutedMoveAbs.Execute := FALSE;
				WorkZone.Step := WAIT;
			END_IF

	END_CASE

	WorkZone.Command();
	WorkZone.RoutedMoveAbs();
	WorkZone.TrgEnable();
	WorkZone.TrgGetInfo();
END_ACTION
```

#### ActWorkStation1.st
```iecst
ACTION ActWorkStation1:

	CASE WorkStation1.Step OF
		WAIT:
			WorkStation1.ElasticMoveAbs.Execute := FALSE;

			IF WorkStation1.TrgEnable.EventCount > 0 THEN
				gStation1ReadyForShuttle := FALSE;
				WorkStation1.TrgGetInfo.Execute := TRUE;
				WorkStation1.Step := DIRECTION_CHECK;
			END_IF

		DIRECTION_CHECK:
			IF WorkStation1.TrgGetInfo.TrgPointInfo.Event = mcACPTRAK_TP_PASSED_POSITIVE THEN
				WorkStation1.Shuttle := WorkStation1.TrgGetInfo.TrgPointInfo.Axis;

				FOR i := 1 TO gMAX_SHUTTLE_CNT DO
					IF WorkStation1.Shuttle.controlif = gShuttleList[i].Axis.controlif THEN
						gShuttleList[i].State := AT_STATION_1;
					END_IF
				END_FOR

				WorkStation1.TrgGetInfo.Execute := FALSE;
				WorkStation1.Step := PROCESS;
			ELSE
				WorkStation1.TrgGetInfo.Execute := FALSE;
				WorkStation1.Step := WAIT;
			END_IF

		PROCESS:
			WorkStation1.Timer.PT := T#2s;
			WorkStation1.Timer.IN := TRUE;

			IF WorkStation1.Timer.Q  AND WorkStation2.ReadyForShuttle THEN
				WorkStation1.Timer.IN := FALSE;
				WorkStation1.Step := SEND_SHUTTLE;
			END_IF

		SEND_SHUTTLE:
			WorkStation1.ElasticMoveAbs.Axis := ADR(WorkStation1.Shuttle);
			WorkStation1.ElasticMoveAbs.Position := 0.99;
			WorkStation1.ElasticMoveAbs.Velocity := gTrakAsm.Parameter.Velocity;
			WorkStation1.ElasticMoveAbs.Acceleration := gTrakAsm.Parameter.Acceleration;
			WorkStation1.ElasticMoveAbs.Deceleration := gTrakAsm.Parameter.Deceleration;
			WorkStation1.ElasticMoveAbs.Jerk := 0.0;
			WorkStation1.ElasticMoveAbs.BufferMode := mcABORTING;
			WorkStation1.ElasticMoveAbs.Execute := TRUE;

			FOR i := 1 TO gMAX_SHUTTLE_CNT DO
				IF WorkStation1.Shuttle.controlif = gShuttleList[i].Axis.controlif THEN
					gShuttleList[i].State := RTE_TO_STATION_2;
				END_IF
			END_FOR

			gStation1ReadyForShuttle := TRUE;
			WorkStation2.ReadyForShuttle := FALSE;
			WorkStation1.Step := WAIT;

	END_CASE

	gStation1EventCount := WorkStation1.TrgEnable.EventCount;

	WorkStation1.ElasticMoveAbs();
	WorkStation1.TrgEnable();
	WorkStation1.TrgGetInfo();
	WorkStation1.Timer();
END_ACTION
```

#### ActWorkStation2.st
```iecst
ACTION ActWorkStation2:

	CASE WorkStation2.Step OF
		WAIT:
			WorkStation2.ElasticMoveAbs.Execute := FALSE;

			IF WorkStation2.TrgEnable.EventCount > 0 THEN
				WorkStation2.TrgGetInfo.Execute := TRUE;
				WorkStation2.Step := DIRECTION_CHECK;
			END_IF

		DIRECTION_CHECK:
			IF WorkStation2.TrgGetInfo.TrgPointInfo.Event = mcACPTRAK_TP_PASSED_POSITIVE THEN
				WorkStation2.Shuttle := WorkStation2.TrgGetInfo.TrgPointInfo.Axis;

				FOR i := 1 TO gMAX_SHUTTLE_CNT DO
					IF WorkStation2.Shuttle.controlif = gShuttleList[i].Axis.controlif THEN
						gShuttleList[i].State := AT_STATION_2;
					END_IF
				END_FOR

				WorkStation2.TrgGetInfo.Execute := FALSE;
				WorkStation2.Step := PROCESS;
			ELSE
				WorkStation2.TrgGetInfo.Execute := FALSE;
				WorkStation2.Step := WAIT;
			END_IF

		PROCESS:
			WorkStation2.Timer.PT := T#2s;
			WorkStation2.Timer.IN := TRUE;

			IF WorkStation2.Timer.Q AND WorkStation3.ReadyForShuttle THEN
				WorkStation2.Timer.IN := FALSE;
				WorkStation2.Step := SEND_SHUTTLE;
			END_IF

		SEND_SHUTTLE:
			WorkStation2.ElasticMoveAbs.Axis := ADR(WorkStation2.Shuttle);
			WorkStation2.ElasticMoveAbs.Position := 1.485;
			WorkStation2.ElasticMoveAbs.Velocity := gTrakAsm.Parameter.Velocity;
			WorkStation2.ElasticMoveAbs.Acceleration := gTrakAsm.Parameter.Acceleration;
			WorkStation2.ElasticMoveAbs.Deceleration := gTrakAsm.Parameter.Deceleration;
			WorkStation2.ElasticMoveAbs.Jerk := 0.0;
			WorkStation2.ElasticMoveAbs.BufferMode := mcABORTING;
			WorkStation2.ElasticMoveAbs.Execute := TRUE;

			FOR i := 1 TO gMAX_SHUTTLE_CNT DO
				IF WorkStation2.Shuttle.controlif = gShuttleList[i].Axis.controlif THEN
					gShuttleList[i].State := RTE_TO_STATION_3;
				END_IF
			END_FOR

			gStation2ReadyForShuttle := TRUE;
			WorkStation3.ReadyForShuttle := FALSE;
			WorkStation2.Step := WAIT;

	END_CASE

	WorkStation2.ElasticMoveAbs();
	WorkStation2.TrgEnable();
	WorkStation2.TrgGetInfo();
	WorkStation2.Timer();
END_ACTION
```

#### ActWorkStation3.st
```iecst
ACTION ActWorkStation3:

	CASE WorkStation3.Step OF
		WAIT:
			WorkStation3.ElasticMoveAbs.Execute := FALSE;

			IF WorkStation3.TrgEnable.EventCount > 0 THEN
				WorkStation3.TrgGetInfo.Execute := TRUE;
				WorkStation3.Step := DIRECTION_CHECK;
			END_IF

		DIRECTION_CHECK:
			IF WorkStation3.TrgGetInfo.TrgPointInfo.Event = mcACPTRAK_TP_PASSED_POSITIVE THEN
				WorkStation3.Shuttle := WorkStation3.TrgGetInfo.TrgPointInfo.Axis;

				FOR i := 1 TO gMAX_SHUTTLE_CNT DO
					IF WorkStation3.Shuttle.controlif = gShuttleList[i].Axis.controlif THEN
						gShuttleList[i].State := AT_STATION_3;
					END_IF
				END_FOR

				WorkStation3.TrgGetInfo.Execute := FALSE;
				WorkStation3.Step := PROCESS;
			ELSE
				WorkStation3.TrgGetInfo.Execute := FALSE;
				WorkStation3.Step := WAIT;
			END_IF

		PROCESS:
			WorkStation3.Timer.PT := T#2s;
			WorkStation3.Timer.IN := TRUE;

			IF WorkStation3.Timer.Q AND WorkStation4.ReadyForShuttle THEN
				WorkStation3.Timer.IN := FALSE;
				WorkStation3.Step := SEND_SHUTTLE;
			END_IF

		SEND_SHUTTLE:
			WorkStation3.ElasticMoveAbs.Axis := ADR(WorkStation3.Shuttle);
			WorkStation3.ElasticMoveAbs.Position := 1.98;
			WorkStation3.ElasticMoveAbs.Velocity := gTrakAsm.Parameter.Velocity;
			WorkStation3.ElasticMoveAbs.Acceleration := gTrakAsm.Parameter.Acceleration;
			WorkStation3.ElasticMoveAbs.Deceleration := gTrakAsm.Parameter.Deceleration;
			WorkStation3.ElasticMoveAbs.Jerk := 0.0;
			WorkStation3.ElasticMoveAbs.BufferMode := mcABORTING;
			WorkStation3.ElasticMoveAbs.Execute := TRUE;

			FOR i := 1 TO gMAX_SHUTTLE_CNT DO
				IF WorkStation3.Shuttle.controlif = gShuttleList[i].Axis.controlif THEN
					gShuttleList[i].State := RTE_TO_STATION_4;
				END_IF
			END_FOR

			gStation3ReadyForShuttle := TRUE;
			WorkStation4.ReadyForShuttle := FALSE;
			WorkStation3.Step := WAIT;

	END_CASE

	WorkStation3.ElasticMoveAbs();
	WorkStation3.TrgEnable();
	WorkStation3.TrgGetInfo();
	WorkStation3.Timer();
END_ACTION
```

#### ActWorkStation4.st
```iecst
ACTION ActWorkStation4:

	CASE WorkStation4.Step OF
		WAIT:
			WorkStation4.RoutedMoveAbs.Execute := FALSE;

			IF WorkStation4.TrgEnable.EventCount > 0 THEN
				WorkStation4.TrgGetInfo.Execute := TRUE;
				WorkStation4.Step := DIRECTION_CHECK;
			END_IF

		DIRECTION_CHECK:
			IF WorkStation4.TrgGetInfo.TrgPointInfo.Event = mcACPTRAK_TP_PASSED_POSITIVE THEN
				WorkStation4.Shuttle := WorkStation4.TrgGetInfo.TrgPointInfo.Axis;

				FOR i := 1 TO gMAX_SHUTTLE_CNT DO
					IF WorkStation4.Shuttle.controlif = gShuttleList[i].Axis.controlif THEN
						gShuttleList[i].State := AT_STATION_4;
					END_IF
				END_FOR

				WorkStation4.TrgGetInfo.Execute := FALSE;
				WorkStation4.Step := PROCESS;
			ELSE
				WorkStation4.TrgGetInfo.Execute := FALSE;
				WorkStation4.Step := WAIT;
			END_IF

		PROCESS:
			WorkStation4.Timer.PT := T#2s;
			WorkStation4.Timer.IN := TRUE;

			IF WorkStation4.Timer.Q THEN
				WorkStation4.Timer.IN := FALSE;
				WorkStation4.Step := SEND_SHUTTLE;
			END_IF

		SEND_SHUTTLE:
			WorkStation4.RoutedMoveAbs.Axis := ADR(WorkStation4.Shuttle);
			WorkStation4.RoutedMoveAbs.Sector := ADR(SectorBuffer);
			WorkStation4.RoutedMoveAbs.Position := 0.2;
			WorkStation4.RoutedMoveAbs.Velocity := gTrakAsm.Parameter.Velocity;
			WorkStation4.RoutedMoveAbs.Acceleration := gTrakAsm.Parameter.Acceleration;
			WorkStation4.RoutedMoveAbs.Deceleration := gTrakAsm.Parameter.Deceleration;
			WorkStation4.RoutedMoveAbs.Jerk := 0.0;
			WorkStation4.RoutedMoveAbs.BufferMode := mcABORTING;
			WorkStation4.RoutedMoveAbs.Execute := TRUE;

			FOR i := 1 TO gMAX_SHUTTLE_CNT DO
				IF WorkStation4.Shuttle.controlif = gShuttleList[i].Axis.controlif THEN
					gShuttleList[i].State := RTE_TO_BUFFER;
				END_IF
			END_FOR

			gStation4ReadyForShuttle := TRUE;
			WorkStation4.Step := WAIT;

	END_CASE

	WorkStation4.TrgEnable();
	WorkStation4.TrgGetInfo();
	WorkStation4.RoutedMoveAbs();
	WorkStation4.Timer();
END_ACTION
```

#### ActThroughputStation.st
```iecst
ACTION ActThroughputStation:
	IF ThroughputTimer.Q THEN
		ThroughputTimer.IN := FALSE;
		CurrentThroughput := ThroughputCounter;
		ThroughputCounter := 0;
	ELSIF NOT ThroughputTimer.IN THEN
		ThroughputTimer.IN := TRUE;
	END_IF

	CASE ThroughputStation.Step OF
		WAIT:
			ThroughputStation.RoutedMoveAbs.Execute := FALSE;
			ThroughputStation.Timer.PT := MAINTENANCE_TIMER_LENGTH;
			ThroughputStation.Timer.IN := TRUE;

			IF ThroughputStation.Timer.Q AND ThroughputStation.TrgEnable.EventCount > 0 THEN
				ThroughputStation.Timer.IN := FALSE;
				ThroughputStation.TrgGetInfo.Execute := TRUE;
				ThroughputStation.Step := DIRECTION_CHECK;
			ELSIF NOT ThroughputStation.Timer.Q AND ThroughputStation.TrgEnable.EventCount > 0 THEN
				ThroughputStation.TrgGetInfo.Execute := TRUE;
				ThroughputStation.Step := DO_NOTHING;
			END_IF

		DO_NOTHING:
			IF ThroughputStation.TrgGetInfo.Done THEN
				ThroughputStation.TrgGetInfo.Execute := FALSE;
				ThroughputCounter := ThroughputCounter + 1;
				ThroughputStation.Step := WAIT;
			END_IF

		DIRECTION_CHECK:
			ThroughputStation.Shuttle := ThroughputStation.TrgGetInfo.TrgPointInfo.Axis;
			ThroughputStation.TrgGetInfo.Execute := FALSE;
			ThroughputCounter := ThroughputCounter + 1;
			ThroughputStation.Step := SEND_SHUTTLE;

		SEND_SHUTTLE:
			ThroughputStation.RoutedMoveAbs.Axis := ADR(ThroughputStation.Shuttle);
			ThroughputStation.RoutedMoveAbs.Sector := ADR(SectorMaintenancePoint);
			ThroughputStation.RoutedMoveAbs.Position := 0.33;
			ThroughputStation.RoutedMoveAbs.Velocity := gTrakAsm.Parameter.Velocity;
			ThroughputStation.RoutedMoveAbs.Acceleration := gTrakAsm.Parameter.Acceleration;
			ThroughputStation.RoutedMoveAbs.Deceleration := gTrakAsm.Parameter.Deceleration;
			ThroughputStation.RoutedMoveAbs.Jerk := 0.0;
			ThroughputStation.RoutedMoveAbs.BufferMode := mcABORTING;
			ThroughputStation.RoutedMoveAbs.Execute := TRUE;

			FOR i := 1 TO gMAX_SHUTTLE_CNT DO
				IF ThroughputStation.Shuttle.controlif = gShuttleList[i].Axis.controlif THEN
					gShuttleList[i].State := RTE_TO_MAINT;
				END_IF
			END_FOR

			ThroughputStation.Step := WAIT;

	END_CASE

	ThroughputStation.RoutedMoveAbs();
	ThroughputStation.TrgEnable();
	ThroughputStation.TrgGetInfo();
	ThroughputStation.Timer();
END_ACTION
```

#### ActMaintenanceStation.st
```iecst
ACTION ActMaintenanceStation:

	CASE MaintenanceStation.Step OF
		WAIT:
			MaintenanceStation.RoutedMoveAbs.Execute := FALSE;

			IF MaintenanceStation.TrgEnable.EventCount > 0 THEN
				MaintenanceStation.TrgGetInfo.Execute := TRUE;
				MaintenanceStation.Step := DIRECTION_CHECK;
			END_IF

		DIRECTION_CHECK:
			IF MaintenanceStation.TrgGetInfo.TrgPointInfo.Event = mcACPTRAK_TP_PASSED_POSITIVE THEN
				MaintenanceStation.Shuttle := MaintenanceStation.TrgGetInfo.TrgPointInfo.Axis;

				FOR i := 1 TO gMAX_SHUTTLE_CNT DO
					IF MaintenanceStation.Shuttle.controlif = gShuttleList[i].Axis.controlif THEN
						gShuttleList[i].State := AT_MAINT;
					END_IF
				END_FOR

				MaintenanceStation.TrgGetInfo.Execute := FALSE;
				MaintenanceStation.Step := PROCESS;
			ELSE
				MaintenanceStation.TrgGetInfo.Execute := FALSE;
				MaintenanceStation.Step := WAIT;
			END_IF

		PROCESS:
			MaintenanceStation.Timer.PT := T#5s;
			MaintenanceStation.Timer.IN := TRUE;

			IF MaintenanceStation.Timer.Q THEN
				MaintenanceStation.Timer.IN := FALSE;
				MaintenanceStation.Step := SEND_SHUTTLE;
			END_IF

		SEND_SHUTTLE:
			MaintenanceStation.RoutedMoveAbs.Axis := ADR(MaintenanceStation.Shuttle);
			MaintenanceStation.RoutedMoveAbs.Sector := ADR(SectorBuffer);
			MaintenanceStation.RoutedMoveAbs.Position := 0.2;
			MaintenanceStation.RoutedMoveAbs.Velocity := gTrakAsm.Parameter.Velocity;
			MaintenanceStation.RoutedMoveAbs.Acceleration := gTrakAsm.Parameter.Acceleration;
			MaintenanceStation.RoutedMoveAbs.Deceleration := gTrakAsm.Parameter.Deceleration;
			MaintenanceStation.RoutedMoveAbs.Jerk := 0.0;
			MaintenanceStation.RoutedMoveAbs.BufferMode := mcABORTING;
			MaintenanceStation.RoutedMoveAbs.Execute := TRUE;

			FOR i := 1 TO gMAX_SHUTTLE_CNT DO
				IF MaintenanceStation.Shuttle.controlif = gShuttleList[i].Axis.controlif THEN
					gShuttleList[i].State := RTE_TO_BUFFER;
				END_IF
			END_FOR

			MaintenanceStation.Step := WAIT;

	END_CASE

	MaintenanceStation.RoutedMoveAbs();
	MaintenanceStation.TrgEnable();
	MaintenanceStation.TrgGetInfo();
	MaintenanceStation.Timer();
END_ACTION
```

### Program Logical/BufferZone (IEC)

#### Variables.var
```iecst
(*Function blocks*)
VAR
	RoutedMoveAbs : MC_BR_RoutedMoveAbs_AcpTrak;
	TrgEnable : MC_BR_TrgPointEnable_AcpTrak;
	TrgGetInfo : MC_BR_TrgPointGetInfo_AcpTrak;
END_VAR
(*Enumerations*)
VAR
	Step : ProcessPointStateEnum;
END_VAR
(*Variables*)
VAR
	Shuttle : McAxisType;
	i : UINT;
	ShuttleIndex : UINT;
	ShuttlesToStation1 : UINT;
END_VAR
(*Constants*)
```

#### Main.st
```iecst
PROGRAM _INIT
	TrgGetInfo.ProcessPoint := ADR(PPBuffer);
	TrgEnable.ProcessPoint := ADR(PPBuffer);
	TrgEnable.Enable := TRUE;

	TrgEnable();
	TrgGetInfo();
END_PROGRAM

PROGRAM _CYCLIC
	CASE Step OF
		WAIT:
			RoutedMoveAbs.Execute := FALSE;

			ShuttlesToStation1 := 0;
			FOR i := 1 TO gMAX_SHUTTLE_CNT DO
				IF gShuttleList[i].State = RTE_TO_STATION_1 THEN
					ShuttlesToStation1 := ShuttlesToStation1 + 1;
				END_IF
			END_FOR

			IF TrgEnable.EventCount > 0 AND ShuttlesToStation1 < gMAX_SHUTTLES_TO_STATION_1 THEN
				 TrgGetInfo.Execute := TRUE;
				 Step := DIRECTION_CHECK;
			END_IF

		DIRECTION_CHECK:
			IF TrgGetInfo.TrgPointInfo.Event = mcACPTRAK_TP_PASSED_POSITIVE THEN
				Shuttle :=  TrgGetInfo.TrgPointInfo.Axis;

				FOR i := 1 TO gMAX_SHUTTLE_CNT DO
					IF  Shuttle.controlif = gShuttleList[i].Axis.controlif THEN
						gShuttleList[i].State := AT_BUFFER;
						ShuttleIndex := i;
					END_IF
				END_FOR

				TrgGetInfo.Execute := FALSE;
				Step := SEND_SHUTTLE;
			ELSE
				TrgGetInfo.Execute := FALSE;
				Step := WAIT;
			END_IF

		SEND_SHUTTLE:
			RoutedMoveAbs.Axis := ADR( Shuttle);
			RoutedMoveAbs.Sector := ADR(SectorWorkZone);
			RoutedMoveAbs.Position := gPROCESS_POINT_LOCATIONS.WORK_ZONE;
			RoutedMoveAbs.Velocity := gTrakAsm.Parameter.Velocity;
			RoutedMoveAbs.Acceleration := gTrakAsm.Parameter.Acceleration;
			RoutedMoveAbs.Deceleration := gTrakAsm.Parameter.Deceleration;
			RoutedMoveAbs.Jerk := 0.0;
			RoutedMoveAbs.BufferMode := mcABORTING;
			RoutedMoveAbs.Execute := TRUE;

			gShuttleList[ShuttleIndex].State := RTE_TO_STATION_1;

			Step := WAIT;

	END_CASE

	RoutedMoveAbs();
	TrgEnable();
	TrgGetInfo();
END_PROGRAM

PROGRAM _EXIT
	(* Insert code here *)

END_PROGRAM
```

### Program Logical/WorkZone (IEC)

#### Variables.var
```iecst
(*Function blocks*)
VAR
	Command : MC_BR_BarrierCommand_AcpTrak;
	RoutedMoveAbs : MC_BR_RoutedMoveAbs_AcpTrak;
	TrgEnable : MC_BR_TrgPointEnable_AcpTrak;
	TrgGetInfo : MC_BR_TrgPointGetInfo_AcpTrak;
END_VAR
(*Enumerations*)
VAR
	Step : ProcessPointStateEnum;
END_VAR
(*Variables*)
VAR
	Shuttle : McAxisType;
	i : UINT;
END_VAR
(*Constants*)
```

#### Main.st
```iecst
PROGRAM _INIT
	TrgGetInfo.ProcessPoint := ADR(PPStation0TrgPoint);
	TrgEnable.ProcessPoint := ADR(PPStation0TrgPoint);
	TrgEnable.Enable := TRUE;
	Command.ProcessPoint := ADR(PPStation0);
	Command.Command := mcACPTRAK_BARRIER_CLOSE;
	Command.Execute := TRUE;

	TrgGetInfo();
	TrgEnable();
	Command();
END_PROGRAM

PROGRAM _CYCLIC
	CASE Step OF
		WAIT:
			Command.Command := mcACPTRAK_BARRIER_CLOSE;
			Command.Execute := TRUE;

			IF TrgEnable.EventCount > 0 AND gStation1ReadyForShuttle THEN
				Command.Execute := FALSE;
				TrgGetInfo.Execute := TRUE;
				Step := DIRECTION_CHECK;
			END_IF

		DIRECTION_CHECK:
			IF TrgGetInfo.TrgPointInfo.Event = mcACPTRAK_TP_PASSED_POSITIVE THEN
				Shuttle := TrgGetInfo.TrgPointInfo.Axis;
				TrgGetInfo.Execute := FALSE;
				Step := PROCESS;
			ELSE
				TrgGetInfo.Execute := FALSE;
				Step := WAIT;
			END_IF

		PROCESS:
			IF gStation1EventCount = 0 THEN
				Step := SEND_SHUTTLE;
			END_IF

		SEND_SHUTTLE:
			RoutedMoveAbs.Axis := ADR(Shuttle);
			RoutedMoveAbs.Sector := ADR(SectorWorkZone);
			RoutedMoveAbs.Position := gPROCESS_POINT_LOCATIONS.WORK_STATION1;
			RoutedMoveAbs.Velocity := gTrakAsm.Parameter.Velocity;
			RoutedMoveAbs.Acceleration := gTrakAsm.Parameter.Acceleration;
			RoutedMoveAbs.Deceleration := gTrakAsm.Parameter.Deceleration;
			RoutedMoveAbs.Jerk := 0.0;
			RoutedMoveAbs.BufferMode := mcABORTING;
			RoutedMoveAbs.Execute := TRUE;

			Command.Command := mcACPTRAK_BARRIER_ADD_TICKETS;
			Command.AdvancedParameters.TicketCount := 1;
			Command.Execute := TRUE;

			IF Command.Done THEN
				gStation1ReadyForShuttle := FALSE;
				Command.Execute := FALSE;
				RoutedMoveAbs.Execute := FALSE;
				Step := WAIT;
			END_IF

	END_CASE

	Command();
	RoutedMoveAbs();
	TrgEnable();
	TrgGetInfo();
END_PROGRAM

PROGRAM _EXIT
	(* Insert code here *)

END_PROGRAM
```

### Program Logical/WorkStation1 (IEC)

#### Main.st
```iecst
PROGRAM _INIT
	TrgGetInfo.ProcessPoint := ADR(PPStation1);
	TrgEnable.ProcessPoint := ADR(PPStation1);
	TrgEnable.Enable := TRUE;

	TrgGetInfo();
	TrgEnable();
END_PROGRAM

PROGRAM _CYCLIC
	CASE Step OF
		WAIT:
			ElasticMoveAbs.Execute := FALSE;

			IF TrgEnable.EventCount > 0 THEN
				gStation1ReadyForShuttle := FALSE;
				TrgGetInfo.Execute := TRUE;
				Step := DIRECTION_CHECK;
			END_IF

		DIRECTION_CHECK:
			IF TrgGetInfo.TrgPointInfo.Event = mcACPTRAK_TP_PASSED_POSITIVE THEN
				Shuttle := TrgGetInfo.TrgPointInfo.Axis;

				FOR i := 1 TO gMAX_SHUTTLE_CNT DO
					IF Shuttle.controlif = gShuttleList[i].Axis.controlif THEN
						gShuttleList[i].State := AT_STATION_1;
						ShuttleIndex := i;
					END_IF
				END_FOR

				TrgGetInfo.Execute := FALSE;
				Step := PROCESS;
			ELSE
				TrgGetInfo.Execute := FALSE;
				Step := WAIT;
			END_IF

		PROCESS:
			Timer.PT := gPROCESS_TIMER_LENGTH;
			Timer.IN := TRUE;

			IF Timer.Q  AND gStation2ReadyForShuttle THEN
				Timer.IN := FALSE;
				Step := SEND_SHUTTLE;
			END_IF

		SEND_SHUTTLE:
			ElasticMoveAbs.Axis := ADR(Shuttle);
			ElasticMoveAbs.Position := gPROCESS_POINT_LOCATIONS.WORK_STATION2;
			ElasticMoveAbs.Velocity := gTrakAsm.Parameter.Velocity;
			ElasticMoveAbs.Acceleration := gTrakAsm.Parameter.Acceleration;
			ElasticMoveAbs.Deceleration := gTrakAsm.Parameter.Deceleration;
			ElasticMoveAbs.Jerk := 0.0;
			ElasticMoveAbs.BufferMode := mcABORTING;
			ElasticMoveAbs.Execute := TRUE;

			gShuttleList[ShuttleIndex].State := RTE_TO_STATION_2;

			gStation1ReadyForShuttle := TRUE;
			gStation2ReadyForShuttle := FALSE;
			Step := WAIT;

	END_CASE

	gStation1EventCount := TrgEnable.EventCount;

	ElasticMoveAbs();
	TrgEnable();
	TrgGetInfo();
	Timer();
END_PROGRAM

PROGRAM _EXIT
	(* Insert code here *)

END_PROGRAM
```

### Program Logical/WorkStation2 (IEC)

#### Variables.var
```iecst
(*Function blocks*)
VAR
	ElasticMoveAbs : MC_BR_ElasticMoveAbs_AcpTrak;
	TrgEnable : MC_BR_TrgPointEnable_AcpTrak;
	TrgGetInfo : MC_BR_TrgPointGetInfo_AcpTrak;
	Timer : TON;
END_VAR
(*Enumerations*)
VAR
	Step : ProcessPointStateEnum;
END_VAR
(*Variables*)
VAR
	Shuttle : McAxisType;
	i : UINT;
	ShuttleIndex : UINT;
	ShuttlesToStation1 : UINT;
END_VAR
(*Constants*)
```

#### Main.st
```iecst
PROGRAM _INIT
	TrgGetInfo.ProcessPoint := ADR(PPStation2);
	TrgEnable.ProcessPoint := ADR(PPStation2);
	TrgEnable.Enable := TRUE;

	TrgGetInfo();
	TrgEnable();
END_PROGRAM

PROGRAM _CYCLIC
	CASE Step OF
		WAIT:
			ElasticMoveAbs.Execute := FALSE;

			IF TrgEnable.EventCount > 0 THEN
				TrgGetInfo.Execute := TRUE;
				Step := DIRECTION_CHECK;
			END_IF

		DIRECTION_CHECK:
			IF TrgGetInfo.TrgPointInfo.Event = mcACPTRAK_TP_PASSED_POSITIVE THEN
				Shuttle := TrgGetInfo.TrgPointInfo.Axis;

				FOR i := 1 TO gMAX_SHUTTLE_CNT DO
					IF Shuttle.controlif = gShuttleList[i].Axis.controlif THEN
						gShuttleList[i].State := AT_STATION_2;
						ShuttleIndex := i;
					END_IF
				END_FOR

				TrgGetInfo.Execute := FALSE;
				Step := PROCESS;
			ELSE
				TrgGetInfo.Execute := FALSE;
				Step := WAIT;
			END_IF

		PROCESS:
			Timer.PT := gPROCESS_TIMER_LENGTH;
			Timer.IN := TRUE;

			IF Timer.Q AND gStation3ReadyForShuttle THEN
				Timer.IN := FALSE;
				Step := SEND_SHUTTLE;
			END_IF

		SEND_SHUTTLE:
			ElasticMoveAbs.Axis := ADR(Shuttle);
			ElasticMoveAbs.Position := gPROCESS_POINT_LOCATIONS.WORK_STATION3;
			ElasticMoveAbs.Velocity := gTrakAsm.Parameter.Velocity;
			ElasticMoveAbs.Acceleration := gTrakAsm.Parameter.Acceleration;
			ElasticMoveAbs.Deceleration := gTrakAsm.Parameter.Deceleration;
			ElasticMoveAbs.Jerk := 0.0;
			ElasticMoveAbs.BufferMode := mcABORTING;
			ElasticMoveAbs.Execute := TRUE;

			gShuttleList[ShuttleIndex].State := RTE_TO_STATION_3;

			gStation2ReadyForShuttle := TRUE;
			gStation3ReadyForShuttle := FALSE;
			Step := WAIT;

	END_CASE

	ElasticMoveAbs();
	TrgEnable();
	TrgGetInfo();
	Timer();
END_PROGRAM

PROGRAM _EXIT
	(* Insert code here *)

END_PROGRAM
```

### Program Logical/WorkStation3 (IEC)

#### Variables.var
```iecst
(*Function blocks*)
VAR
	ElasticMoveAbs : MC_BR_ElasticMoveAbs_AcpTrak;
	TrgEnable : MC_BR_TrgPointEnable_AcpTrak;
	TrgGetInfo : MC_BR_TrgPointGetInfo_AcpTrak;
	Timer : TON;
END_VAR
(*Enumerations*)
VAR
	Step : ProcessPointStateEnum;
END_VAR
(*Variables*)
VAR
	Shuttle : McAxisType;
	i : UINT;
	ShuttlesToStation1 : UINT;
END_VAR
(*Constants*)
```

#### Main.st
```iecst
PROGRAM _INIT
	TrgGetInfo.ProcessPoint := ADR(PPStation3);
	TrgEnable.ProcessPoint := ADR(PPStation3);
	TrgEnable.Enable := TRUE;

	TrgGetInfo();
	TrgEnable();
END_PROGRAM

PROGRAM _CYCLIC
	CASE Step OF
		WAIT:
			ElasticMoveAbs.Execute := FALSE;

			IF TrgEnable.EventCount > 0 THEN
				TrgGetInfo.Execute := TRUE;
				Step := DIRECTION_CHECK;
			END_IF

		DIRECTION_CHECK:
			IF TrgGetInfo.TrgPointInfo.Event = mcACPTRAK_TP_PASSED_POSITIVE THEN
				Shuttle := TrgGetInfo.TrgPointInfo.Axis;

				FOR i := 1 TO gMAX_SHUTTLE_CNT DO
					IF Shuttle.controlif = gShuttleList[i].Axis.controlif THEN
						gShuttleList[i].State := AT_STATION_3;
						ShuttleIndex := i;
					END_IF
				END_FOR

				TrgGetInfo.Execute := FALSE;
				Step := PROCESS;
			ELSE
				TrgGetInfo.Execute := FALSE;
				Step := WAIT;
			END_IF

		PROCESS:
			Timer.PT := gPROCESS_TIMER_LENGTH;
			Timer.IN := TRUE;

			IF Timer.Q AND gStation4ReadyForShuttle THEN
				Timer.IN := FALSE;
				Step := SEND_SHUTTLE;
			END_IF

		SEND_SHUTTLE:
			ElasticMoveAbs.Axis := ADR(Shuttle);
			ElasticMoveAbs.Position := gPROCESS_POINT_LOCATIONS.WORK_STATION4;
			ElasticMoveAbs.Velocity := gTrakAsm.Parameter.Velocity;
			ElasticMoveAbs.Acceleration := gTrakAsm.Parameter.Acceleration;
			ElasticMoveAbs.Deceleration := gTrakAsm.Parameter.Deceleration;
			ElasticMoveAbs.Jerk := 0.0;
			ElasticMoveAbs.BufferMode := mcABORTING;
			ElasticMoveAbs.Execute := TRUE;

			gShuttleList[ShuttleIndex].State := RTE_TO_STATION_4;

			gStation3ReadyForShuttle := TRUE;
			gStation4ReadyForShuttle := FALSE;
			Step := WAIT;

	END_CASE

	ElasticMoveAbs();
	TrgEnable();
	TrgGetInfo();
	Timer();
END_PROGRAM

PROGRAM _EXIT
	(* Insert code here *)

END_PROGRAM
```

### Program Logical/WorkStation4 (IEC)

#### Variables.var
```iecst
(*Function blocks*)
VAR
	RoutedMoveAbs : MC_BR_RoutedMoveAbs_AcpTrak;
	TrgEnable : MC_BR_TrgPointEnable_AcpTrak;
	TrgGetInfo : MC_BR_TrgPointGetInfo_AcpTrak;
	Timer : TON;
END_VAR
(*Enumerations*)
VAR
	Step : ProcessPointStateEnum;
END_VAR
(*Variables*)
VAR
	Shuttle : McAxisType;
	i : UINT;
	ShuttleIndex : UINT;
	ShuttlesToStation1 : UINT;
END_VAR
(*Constants*)
```

#### Main.st
```iecst
PROGRAM _INIT
	TrgGetInfo.ProcessPoint := ADR(PPStation4);
	TrgEnable.ProcessPoint := ADR(PPStation4);
	TrgEnable.Enable := TRUE;

	TrgGetInfo();
	TrgEnable();
END_PROGRAM

PROGRAM _CYCLIC
	CASE Step OF
		WAIT:
			RoutedMoveAbs.Execute := FALSE;

			IF TrgEnable.EventCount > 0 THEN
				TrgGetInfo.Execute := TRUE;
				Step := DIRECTION_CHECK;
			END_IF

		DIRECTION_CHECK:
			IF TrgGetInfo.TrgPointInfo.Event = mcACPTRAK_TP_PASSED_POSITIVE THEN
				Shuttle := TrgGetInfo.TrgPointInfo.Axis;

				FOR i := 1 TO gMAX_SHUTTLE_CNT DO
					IF Shuttle.controlif = gShuttleList[i].Axis.controlif THEN
						gShuttleList[i].State := AT_STATION_4;
						ShuttleIndex := i;
					END_IF
				END_FOR

				TrgGetInfo.Execute := FALSE;
				Step := PROCESS;
			ELSE
				TrgGetInfo.Execute := FALSE;
				Step := WAIT;
			END_IF

		PROCESS:
			Timer.PT := gPROCESS_TIMER_LENGTH;
			Timer.IN := TRUE;

			IF Timer.Q THEN
				Timer.IN := FALSE;
				Step := SEND_SHUTTLE;
			END_IF

		SEND_SHUTTLE:
			RoutedMoveAbs.Axis := ADR(Shuttle);
			RoutedMoveAbs.Sector := ADR(SectorBuffer);
			RoutedMoveAbs.Position := gPROCESS_POINT_LOCATIONS.BUFFER;
			RoutedMoveAbs.Velocity := gTrakAsm.Parameter.Velocity;
			RoutedMoveAbs.Acceleration := gTrakAsm.Parameter.Acceleration;
			RoutedMoveAbs.Deceleration := gTrakAsm.Parameter.Deceleration;
			RoutedMoveAbs.Jerk := 0.0;
			RoutedMoveAbs.BufferMode := mcABORTING;
			RoutedMoveAbs.Execute := TRUE;

			gShuttleList[ShuttleIndex].State := RTE_TO_BUFFER;

			gStation4ReadyForShuttle := TRUE;
			Step := WAIT;

	END_CASE

	RoutedMoveAbs();
	TrgEnable();
	TrgGetInfo();
	RoutedMoveAbs();
	Timer();
END_PROGRAM

PROGRAM _EXIT
	(* Insert code here *)

END_PROGRAM
```

### Program Logical/ThroughputStation (IEC)

#### Variables.var
```iecst
(*Function blocks*)
VAR
	RoutedMoveAbs : MC_BR_RoutedMoveAbs_AcpTrak;
	TrgEnable : MC_BR_TrgPointEnable_AcpTrak;
	TrgGetInfo : MC_BR_TrgPointGetInfo_AcpTrak;
	Timer : TON;
END_VAR
(*Enumerations*)
VAR
	Step : ProcessPointStateEnum;
END_VAR
(*Variables*)
VAR
	Shuttle : McAxisType;
	i : UINT;
	ShuttlesToStation1 : UINT;
	ThroughputCounter : INT := 0;
END_VAR
(*Constants*)
VAR CONSTANT
	MAINTENANCE_TIMER_LENGTH : TIME := T#30s;
END_VAR
```

#### Main.st
```iecst
PROGRAM _INIT
	TrgGetInfo.ProcessPoint := ADR(PPThroughput);
	TrgEnable.ProcessPoint := ADR(PPThroughput);
	TrgEnable.Enable := TRUE;

	TrgGetInfo();
	TrgEnable();
END_PROGRAM

PROGRAM _CYCLIC
	IF gThroughputTimer.Q THEN
		gThroughputTimer.IN := FALSE;
		gCurrentThroughput := ThroughputCounter;
		ThroughputCounter := 0;
	ELSIF NOT gThroughputTimer.IN THEN
		gThroughputTimer.IN := TRUE;
	END_IF

	CASE Step OF
		WAIT:
			RoutedMoveAbs.Execute := FALSE;
			Timer.PT := MAINTENANCE_TIMER_LENGTH;
			Timer.IN := TRUE;

			IF TrgEnable.EventCount > 0 THEN
				TrgGetInfo.Execute := TRUE;
				Step := DIRECTION_CHECK;
			END_IF

		DIRECTION_CHECK:
			IF Timer.Q THEN
				Timer.IN := FALSE;
				Shuttle := TrgGetInfo.TrgPointInfo.Axis;
				TrgGetInfo.Execute := FALSE;
				ThroughputCounter := ThroughputCounter + 1;
				Step := SEND_SHUTTLE;
			ELSE
				TrgGetInfo.Execute := FALSE;
				ThroughputCounter := ThroughputCounter + 1;
				Step := WAIT;
			END_IF

		SEND_SHUTTLE:
			RoutedMoveAbs.Axis := ADR(Shuttle);
			RoutedMoveAbs.Sector := ADR(SectorMaintenancePoint);
			RoutedMoveAbs.Position := gPROCESS_POINT_LOCATIONS.MAINTENANCE_POINT;
			RoutedMoveAbs.Velocity := gTrakAsm.Parameter.Velocity;
			RoutedMoveAbs.Acceleration := gTrakAsm.Parameter.Acceleration;
			RoutedMoveAbs.Deceleration := gTrakAsm.Parameter.Deceleration;
			RoutedMoveAbs.Jerk := 0.0;
			RoutedMoveAbs.BufferMode := mcABORTING;
			RoutedMoveAbs.Execute := TRUE;

			FOR i := 1 TO gMAX_SHUTTLE_CNT DO
				IF Shuttle.controlif = gShuttleList[i].Axis.controlif THEN
					gShuttleList[i].State := RTE_TO_MAINT;
				END_IF
			END_FOR

			Step := WAIT;

	END_CASE

	RoutedMoveAbs();
	TrgEnable();
	TrgGetInfo();
	Timer();
END_PROGRAM

PROGRAM _EXIT
	(* Insert code here *)

END_PROGRAM
```

### Program Logical/MaintenanceStation (IEC)

#### Variables.var
```iecst
(*Function blocks*)
VAR
	RoutedMoveAbs : MC_BR_RoutedMoveAbs_AcpTrak;
	TrgEnable : MC_BR_TrgPointEnable_AcpTrak;
	TrgGetInfo : MC_BR_TrgPointGetInfo_AcpTrak;
	Timer : TON;
END_VAR
(*Enumerations*)
VAR
	Step : ProcessPointStateEnum;
END_VAR
(*Variables*)
VAR
	Shuttle : McAxisType;
	i : UINT;
	ShuttleIndex : UINT;
	ShuttlesToStation1 : UINT;
	ThroughputCounter : INT := 0;
END_VAR
(*Constants*)
VAR CONSTANT
	MAINTENANCE_TIMER_LENGTH : TIME := T#30s;
END_VAR
```

#### Main.st
```iecst
PROGRAM _INIT
	TrgGetInfo.ProcessPoint := ADR(PPMaintenancePoint);
	TrgEnable.ProcessPoint := ADR(PPMaintenancePoint);
	TrgEnable.Enable := TRUE;

	TrgGetInfo();
	TrgEnable();
END_PROGRAM

PROGRAM _CYCLIC
	CASE Step OF
		WAIT:
			RoutedMoveAbs.Execute := FALSE;

			IF TrgEnable.EventCount > 0 THEN
				TrgGetInfo.Execute := TRUE;
				Step := DIRECTION_CHECK;
			END_IF

		DIRECTION_CHECK:
			IF TrgGetInfo.TrgPointInfo.Event = mcACPTRAK_TP_PASSED_POSITIVE THEN
				Shuttle := TrgGetInfo.TrgPointInfo.Axis;

				FOR i := 1 TO gMAX_SHUTTLE_CNT DO
					IF Shuttle.controlif = gShuttleList[i].Axis.controlif THEN
						gShuttleList[i].State := AT_MAINT;
						ShuttleIndex := i;
					END_IF
				END_FOR

				TrgGetInfo.Execute := FALSE;
				Step := PROCESS;
			ELSE
				TrgGetInfo.Execute := FALSE;
				Step := WAIT;
			END_IF

		PROCESS:
			Timer.PT := gMAINTENCANCE_TIMER_LENGTH;
			Timer.IN := TRUE;

			IF Timer.Q THEN
				Timer.IN := FALSE;
				Step := SEND_SHUTTLE;
			END_IF

		SEND_SHUTTLE:
			RoutedMoveAbs.Axis := ADR(Shuttle);
			RoutedMoveAbs.Sector := ADR(SectorBuffer);
			RoutedMoveAbs.Position := gPROCESS_POINT_LOCATIONS.BUFFER;
			RoutedMoveAbs.Velocity := gTrakAsm.Parameter.Velocity;
			RoutedMoveAbs.Acceleration := gTrakAsm.Parameter.Acceleration;
			RoutedMoveAbs.Deceleration := gTrakAsm.Parameter.Deceleration;
			RoutedMoveAbs.Jerk := 0.0;
			RoutedMoveAbs.BufferMode := mcABORTING;
			RoutedMoveAbs.Execute := TRUE;

			gShuttleList[ShuttleIndex].State := RTE_TO_BUFFER;

			Step := WAIT;

	END_CASE

	RoutedMoveAbs();
	TrgEnable();
	TrgGetInfo();
	Timer();
END_PROGRAM

PROGRAM _EXIT
	(* Insert code here *)

END_PROGRAM
```
